# EPICS substitutions: iocs/example_old/exampleApp/Db/posCompEx.substitutions
file positioncompare.template
{
pattern { P, PORT, PLC, PMAC }
		{ P, pmac_S0, 15, 4 }
}
